# EPICS autosave request: ADPvCam/pvcamApp/Db/pvCam_settings.req
file "ADBase_settings.req", P=$(P), R=$(R)
$(P)$(R)GainX
$(P)$(R)GainY
$(P)$(R)Fidget
